// TIA Portal V19 export
DATA_BLOCK "A04_HMI_IDB"   // DB216
AUTHOR : Piemme
FAMILY : System
// stored: InstanceOfName HMI_A04_FB, InstanceOfType FB
"HMI_A04_FB"
   // VAR_OUTPUT
   //    MB4_LpJog : Bool;
   // END_VAR
   // VAR
   //    MB4_Decoder { ExternalAccessible := 'False'; ExternalVisible := 'False'; ExternalWritable := 'False'} : "ButtonsHMIDecoder";
   // END_VAR
BEGIN
END_DATA_BLOCK
